{attribute 'GeneratedUsingTerminal: EL9011--0000'}
{attribute addProperty VendorId "#x00000002"}
{attribute addProperty BoxType "EL9011--0000"}
{attribute addProperty Description "EL9011 End Terminal"}
{attribute addProperty Physics ""}
{attribute addProperty Id "EL9011"}
{attribute addProperty CRC "3596434738"}
{attribute addProperty Size "0"}
TYPE EL9011_D65D3D32 EXTENDS TcoIo.EtcSlaveEndTerminalBase_866C7F0C :
STRUCT
END_STRUCT
END_TYPE

(* stored: Version 1.2.0.0, ProductVersion 3.1.4024.11
   DUT EL9011_D65D3D32: Id {17f1c1df-4650-06c9-0c8a-74feb0dd3811} *)
